// TIA Portal V21 export
TYPE "Std_ParametriMacchina(010102)"
   STRUCT
      Temperatura : Struct
         Online : Real;
         Offline : Real;
      END_STRUCT;
      MinimaTempSteriliz : Struct
         Online : Real;
         Offline : Real;
      END_STRUCT;
      LivelloSerbatoio : Struct
         Online : Real;
         Offline : Real;
      END_STRUCT;
   END_STRUCT;
END_TYPE
